ABB RobotStudio station: ABBPracticalTraining.rsstnx

Station ABBPracticalTraining (saved by RobotStudio 25.2.11220.0)
Controller IRB2600_12_165
  mechanical unit ROB_1: IRB2600_12_165__02, 6 joints, base frame (0, 0, 0) mm
Layout (positions relative to the parent item):
  - IRB2600_12_165__02 [mechanism, from %ABB.RobotStudio.Models.IRB2600%\IRB2600_12_165_G_02.rslib] at (0, 0, 0) mm; joint values [0.2014, 0.0005, -0.0434, 3.1968, -1.5603, -4.4214] (rad or m)
  - table_and_fixture_140 [part] at (667.23, 143.07, 0) mm, size 450 x 350 x 308 mm
  - Tool_suck [mechanism, from ABBPracticalTraining_1\Tool_suck.rslib] at (924.16, 193.52, 1209.24) mm, rotated rx -177.97 ry 3.9 rz -95.01 deg
  - table_and_fixture_141 [part] at (667.23, -206.93, 0) mm, size 450 x 350 x 308 mm
  - 部件_1 [part] at (1287.5, -72.5, 1018.82) mm, rotated rx 0 ry -0.05 rz 0 deg, size 400 x 300 x 200 mm
  - SmartComponent_1 [smart component]
      signals: DI di0
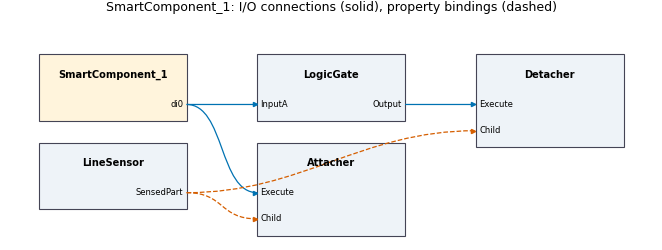
      connections:
        SmartComponent_1.di0 -> LogicGate.InputA
        LogicGate.Output -> Detacher.Execute
        SmartComponent_1.di0 -> Attacher.Execute
        LineSensor.SensedPart => Attacher.Child
        LineSensor.SensedPart => Detacher.Child
    - Attacher [smart component, from Components\Attacher.rslib]
        properties: Parent=Tool_suck; Flange=0; Child=(none); Mount=false; Offset=[0 0 0]; Orientation=[0 0 0]
    - Detacher [smart component, from Components\Detacher.rslib]
        properties: Child=(none); KeepPosition=true
    - LogicGate [smart component, from Components\LogicGate.rslib]
        properties: Operator=NOT; Delay=0
    - LineSensor [smart component, from Components\LineSensor.rslib] at (927.05, 198.04, 1139.45) mm, rotated rx -177.97 ry 3.9 rz -95.01 deg
        properties: Start=[0 0 0.11]; End=[0 0 0.09]; Length=0.02; Radius=0.002; Tag=(none); SenseMultiple=false; SensedPart=(none); SensedPoint=[0 0 0]
      - _sensorPart_ [part], size 4 x 4 x 20 mm
Attachment: Tool_suck is attached to IRB2600_12_165__02 / Link6
Attachment: LineSensor is attached to Tool_suck / TOOL1
Station logic (signal -> signal, property => property):
  IRB2600_12_165.do0 -> SmartComponent_1.di0
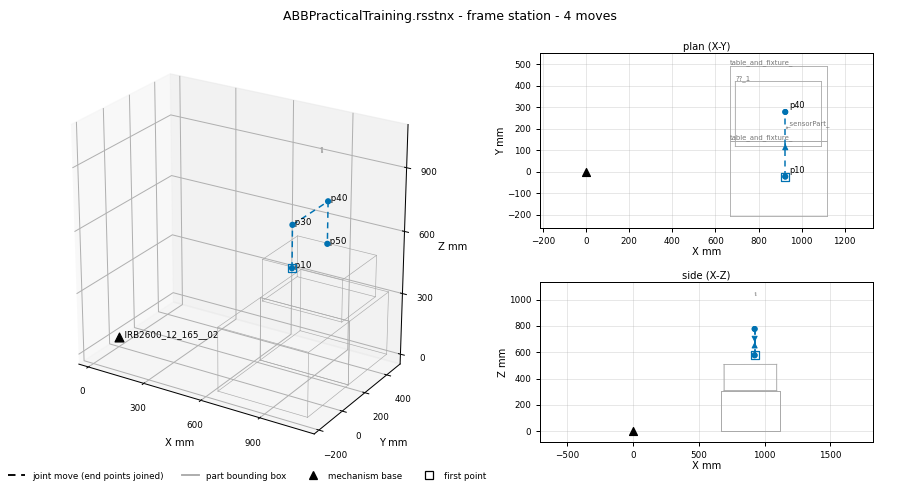
[picture p0: tool path of ABBPracticalTraining.rsstnx in frame station, 4 of 6 moves have a stored position in this frame; points joined in program order, loops and branches not executed]
Targets, tools, work objects and paths stored in the station, written as RAPID:
! task T_ROB1
MODULE CalibData
  PERS tooldata MyTool:=[TRUE,[[31.792631019,0,229.638935148],[0.945518576,0,0.325568154,0]],[1,[0,0,1],[1,0,0,0],0,0,0]];
  TASK PERS wobjdata Workobject_1:=[FALSE,TRUE,"",[[788.717,721.202,308],[0,0,0,1]],[[0,0,0],[1,0,0,0]]];
  PERS tooldata Tool_suck:=[TRUE,[[0,0,70],[1,0,0,0]],[1,[0,0,1],[1,0,0,0],0,0,0]];
ENDMODULE

! task T_ROB1
MODULE MainModule
  CONST robtarget p10:=[[924.16,-22.34,576.5],[0.0370625,-0.674596,0.737188,0.00996895],[-1,2,-4,1],[9E+09,9E+09,9E+09,9E+09,9E+09,9E+09]];
  CONST robtarget p30:=[[924.16,-22.34,776.5],[0.0370629,-0.674596,0.737189,0.00996926],[-1,2,-3,1],[9E+09,9E+09,9E+09,9E+09,9E+09,9E+09]];
  CONST robtarget p40:=[[924.16,277.66,776.5],[0.0370627,-0.674596,0.737188,0.00996888],[0,2,-3,1],[9E+09,9E+09,9E+09,9E+09,9E+09,9E+09]];
  CONST robtarget p50:=[[924.16,277.66,576.5],[0.0370625,-0.674597,0.737188,0.00996883],[0,2,-3,1],[9E+09,9E+09,9E+09,9E+09,9E+09,9E+09]];
  PROC main()
    Reset do0;
    MoveAbsJ il_1\NoEOffs,v1000,z50,tool0;
    MoveJ p10,v1000,z50,tool0;
    Set do0;
    MoveJ p30,v1000,z50,tool0;
    MoveJ p40,v1000,z50,tool0;
    MoveJ p50,v1000,z50,tool0;
    Reset do0;
    MoveAbsJ il_2\NoEOffs,v1000,z50,tool0;
  ENDPROC
ENDMODULE

